// TIA Portal V20 export
TYPE "typeSequenceControlNode"
// stored: Namespace Unit1.Em1
   STRUCT
      jobs { ExternalWritable := 'False'} : "LAF_typeJobs";
      sequence { ExternalWritable := 'False'} : "LAF_typeSequence";
      "step" { ExternalWritable := 'False'} : "LER_typeStep";
      jobInterface { ExternalWritable := 'False'} : "Unit1.Em1.typeSequenceControlNodeJobInterface";
   END_STRUCT;
END_TYPE
